{attribute 'qualified_only'}
{attribute 'strict'}
{attribute 'to_string'}
TYPE TRAFFIC_LIGHT_MODE :
(
	NORMAL,
	BLINKING_YELLOW
);
END_TYPE

(* stored: Version 1.1.0.1
   DUT TRAFFIC_LIGHT_MODE: Id {b620d584-cfa1-4a4e-9931-6f98bba3c0d5} *)
